% RSLogix 500 project IO_Timers.RSS, saved by version 8.30.01.01 %
PROJECT "PROG_01"    % processor: Bul.1763 MicroLogix 1100 Series A %

PROGRAM FILES
  LAD 2   5 rungs

DATA FILES
  O0 OUTPUT  4 elements
  I1 INPUT  6 elements
  S2 STATUS  66 elements
  B3 BINARY  1 elements
  T4 TIMER  1 elements
  C5 COUNTER  1 elements
  R6 CONTROL  1 elements
  N7 INTEGER  1 elements
  F8 FLOAT  1 elements

LADDER 2
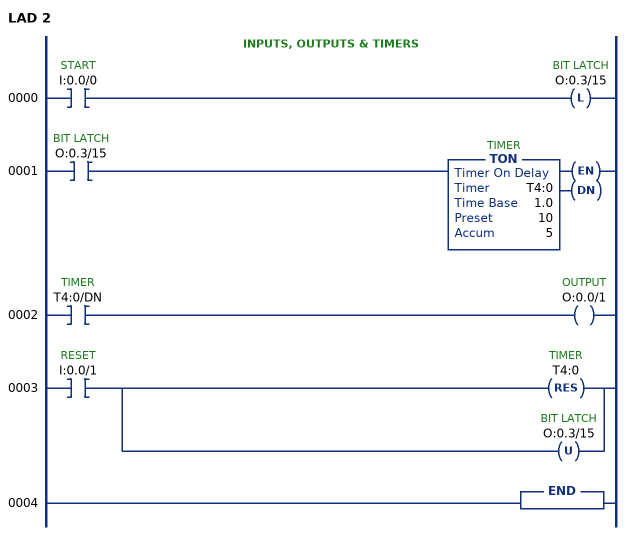
% Rung: 0 %
% TITLE: INPUTS, OUTPUTS & TIMERS %
SOR XIC I:0.0/0 OTL O:0.3/15 EOR
%   I:0.0/0  "START" %
%   O:0.3/15  "BIT LATCH" %
% Rung: 1 %
SOR XIC O:0.3/15 TON T4:0 1.0 10 5 EOR
%   O:0.3/15  "BIT LATCH" %
%   T4:0  "TIMER" %
% Rung: 2 %
SOR XIC T4:0/DN OTE O:0.0/1 EOR
%   T4:0  "TIMER" %
%   O:0.0/1  "OUTPUT" %
% Rung: 3 %  % edit flag set %
SOR XIC I:0.0/1 BST RES T4:0 NXB OTU O:0.3/15 BND EOR
%   I:0.0/1  "RESET" %
%   T4:0  "TIMER" %
%   O:0.3/15  "BIT LATCH" %
% Rung: 4 %
SOR END EOR

REVISION NOTES
  0: Ejemplo de uso de entradas, salidas, variables y temporizador.

DATA TABLE (non-zero values as saved)
DATA T4
% .PRE .ACC %
% T4:0 % 10 5
